PROGRAM MAIN
VAR
	light: bool;
END_VAR

//proj for testing

END_PROGRAM

(* stored: Version 1.1.0.1, ProductVersion 3.1.4026.6
   POU MAIN: Id {443be2ee-236d-4b6a-a245-3675c985b178}, SpecialFunc None *)
